// Mitsubishi GX Works2 project: 20151109(変えた)   PLC: Q03UDV

PROGRAM P1
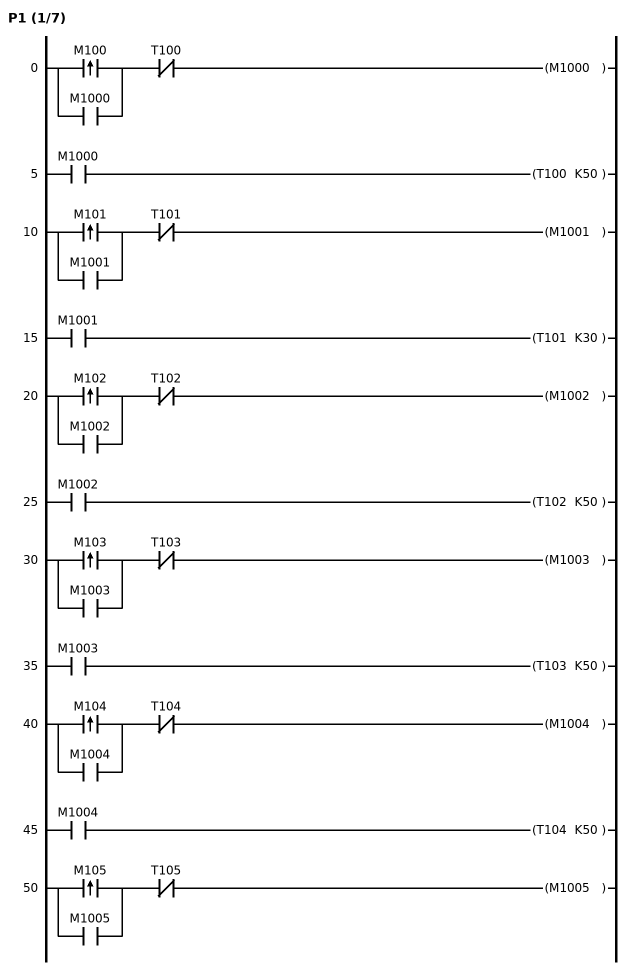
0     LDP     M100
      OR      M1000
      ANI     T100
      OUT     M1000
5     LD      M1000
      OUT     T100 K50
10    LDP     M101
      OR      M1001
      ANI     T101
      OUT     M1001
15    LD      M1001
      OUT     T101 K30
20    LDP     M102
      OR      M1002
      ANI     T102
      OUT     M1002
25    LD      M1002
      OUT     T102 K50
30    LDP     M103
      OR      M1003
      ANI     T103
      OUT     M1003
35    LD      M1003
      OUT     T103 K50
40    LDP     M104
      OR      M1004
      ANI     T104
      OUT     M1004
45    LD      M1004
      OUT     T104 K50
50    LDP     M105
      OR      M1005
      ANI     T105
      OUT     M1005
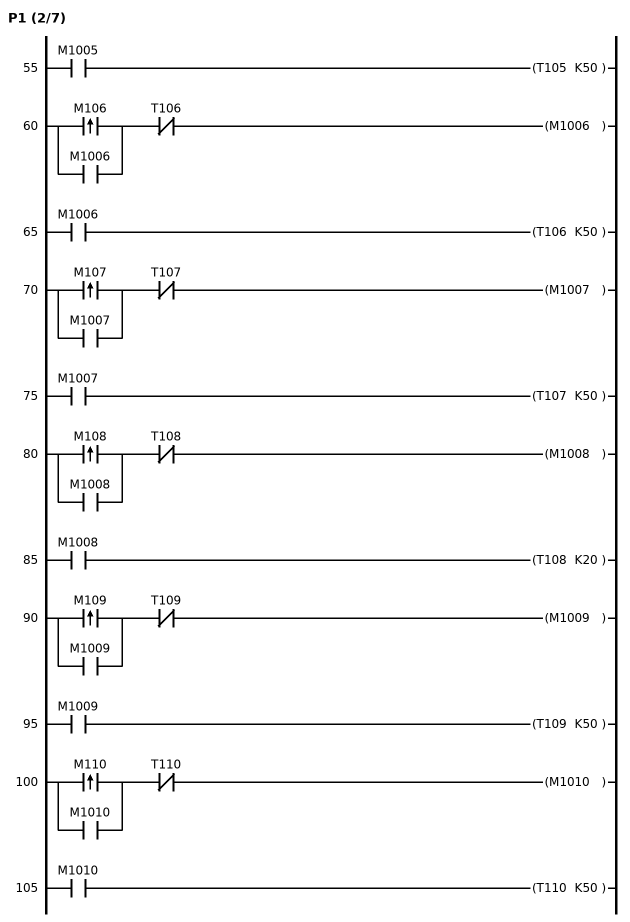
55    LD      M1005
      OUT     T105 K50
60    LDP     M106
      OR      M1006
      ANI     T106
      OUT     M1006
65    LD      M1006
      OUT     T106 K50
70    LDP     M107
      OR      M1007
      ANI     T107
      OUT     M1007
75    LD      M1007
      OUT     T107 K50
80    LDP     M108
      OR      M1008
      ANI     T108
      OUT     M1008
85    LD      M1008
      OUT     T108 K20
90    LDP     M109
      OR      M1009
      ANI     T109
      OUT     M1009
95    LD      M1009
      OUT     T109 K50
100   LDP     M110
      OR      M1010
      ANI     T110
      OUT     M1010
105   LD      M1010
      OUT     T110 K50
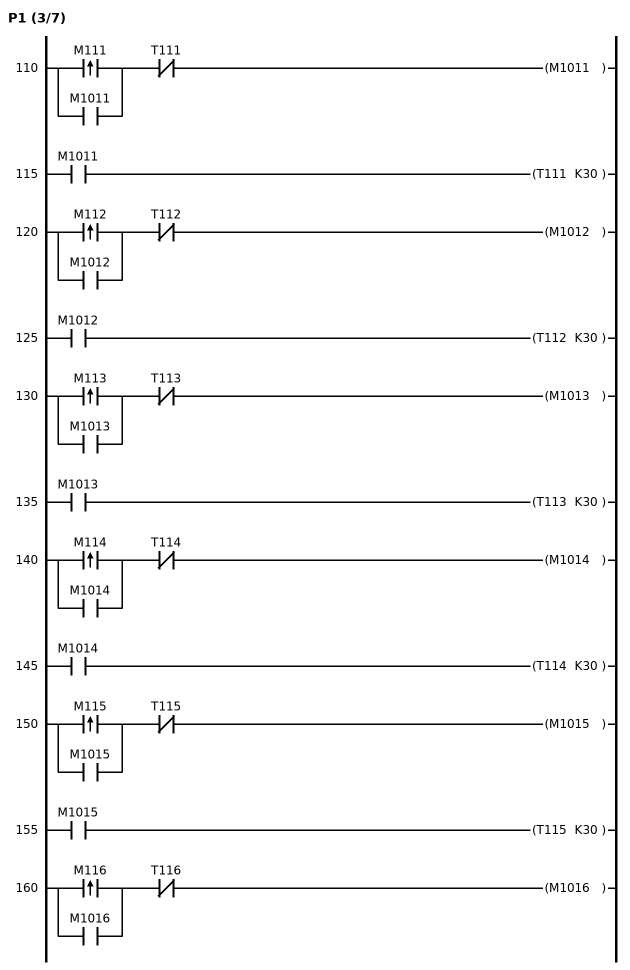
110   LDP     M111
      OR      M1011
      ANI     T111
      OUT     M1011
115   LD      M1011
      OUT     T111 K30
120   LDP     M112
      OR      M1012
      ANI     T112
      OUT     M1012
125   LD      M1012
      OUT     T112 K30
130   LDP     M113
      OR      M1013
      ANI     T113
      OUT     M1013
135   LD      M1013
      OUT     T113 K30
140   LDP     M114
      OR      M1014
      ANI     T114
      OUT     M1014
145   LD      M1014
      OUT     T114 K30
150   LDP     M115
      OR      M1015
      ANI     T115
      OUT     M1015
155   LD      M1015
      OUT     T115 K30
160   LDP     M116
      OR      M1016
      ANI     T116
      OUT     M1016
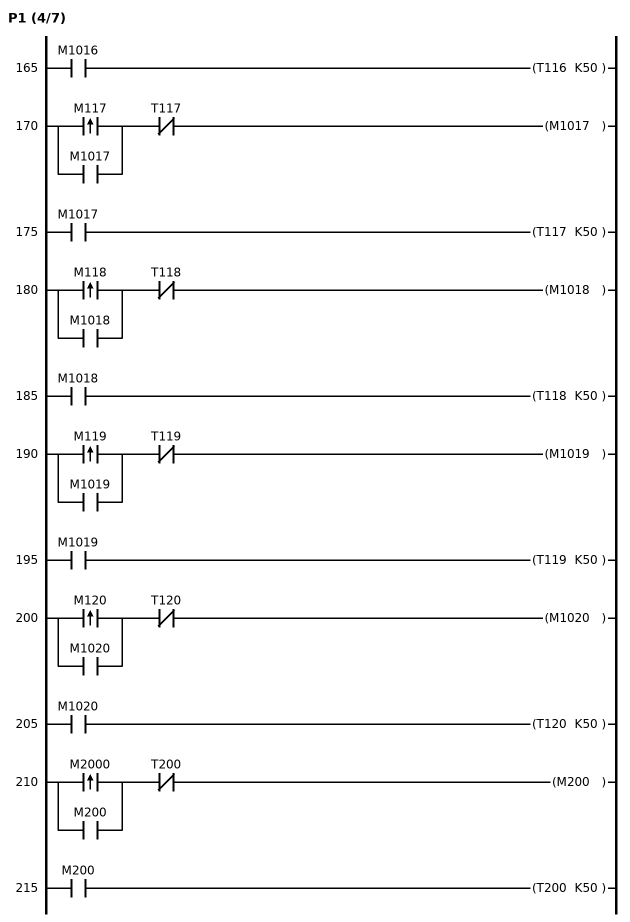
165   LD      M1016
      OUT     T116 K50
170   LDP     M117
      OR      M1017
      ANI     T117
      OUT     M1017
175   LD      M1017
      OUT     T117 K50
180   LDP     M118
      OR      M1018
      ANI     T118
      OUT     M1018
185   LD      M1018
      OUT     T118 K50
190   LDP     M119
      OR      M1019
      ANI     T119
      OUT     M1019
195   LD      M1019
      OUT     T119 K50
200   LDP     M120
      OR      M1020
      ANI     T120
      OUT     M1020
205   LD      M1020
      OUT     T120 K50
210   LDP     M2000
      OR      M200
      ANI     T200
      OUT     M200
215   LD      M200
      OUT     T200 K50
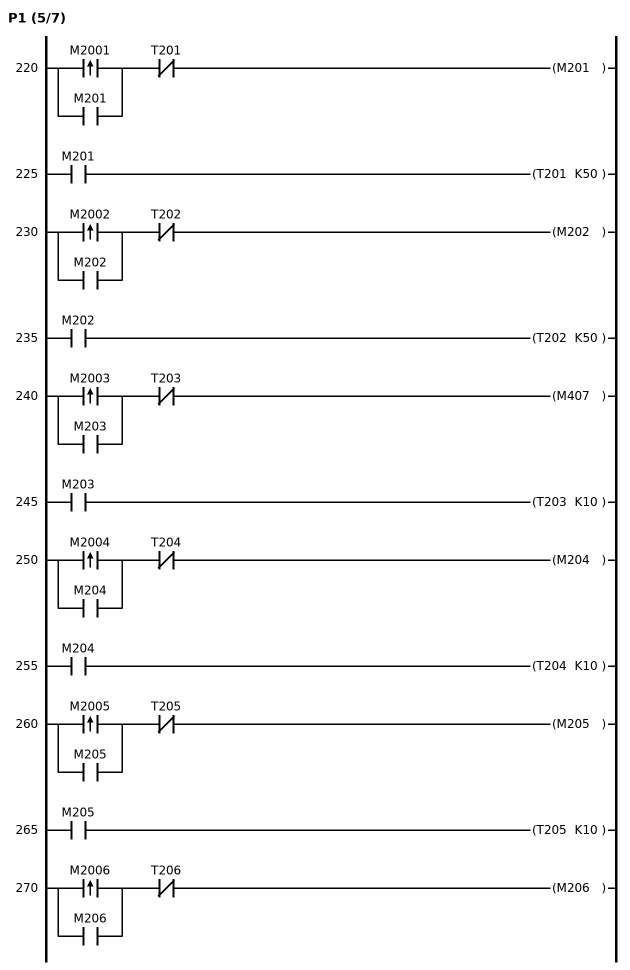
220   LDP     M2001
      OR      M201
      ANI     T201
      OUT     M201
225   LD      M201
      OUT     T201 K50
230   LDP     M2002
      OR      M202
      ANI     T202
      OUT     M202
235   LD      M202
      OUT     T202 K50
240   LDP     M2003
      OR      M203
      ANI     T203
      OUT     M407
245   LD      M203
      OUT     T203 K10
250   LDP     M2004
      OR      M204
      ANI     T204
      OUT     M204
255   LD      M204
      OUT     T204 K10
260   LDP     M2005
      OR      M205
      ANI     T205
      OUT     M205
265   LD      M205
      OUT     T205 K10
270   LDP     M2006
      OR      M206
      ANI     T206
      OUT     M206
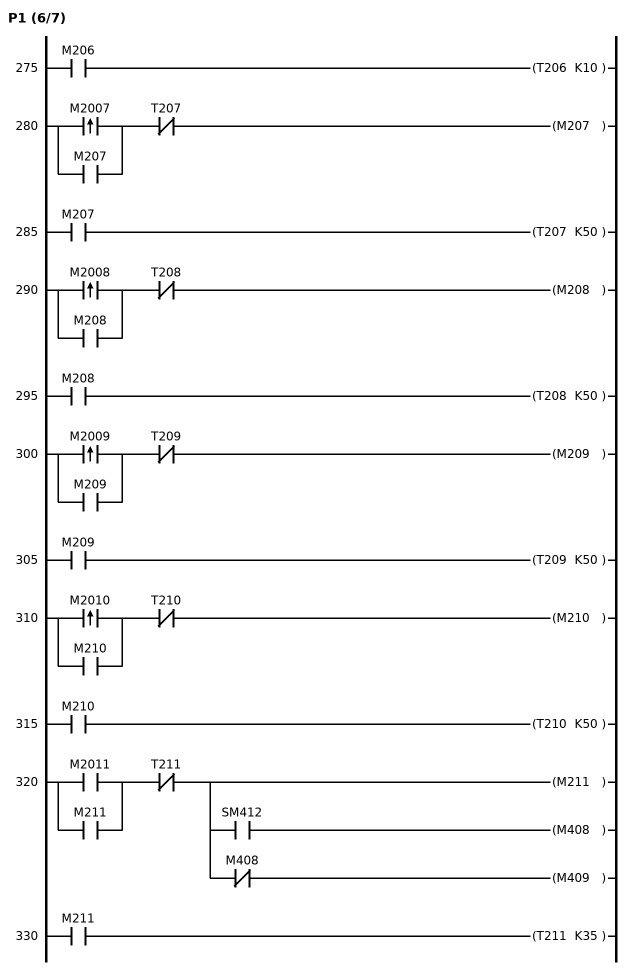
275   LD      M206
      OUT     T206 K10
280   LDP     M2007
      OR      M207
      ANI     T207
      OUT     M207
285   LD      M207
      OUT     T207 K50
290   LDP     M2008
      OR      M208
      ANI     T208
      OUT     M208
295   LD      M208
      OUT     T208 K50
300   LDP     M2009
      OR      M209
      ANI     T209
      OUT     M209
305   LD      M209
      OUT     T209 K50
310   LDP     M2010
      OR      M210
      ANI     T210
      OUT     M210
315   LD      M210
      OUT     T210 K50
320   LD      M2011
      OR      M211
      ANI     T211
      OUT     M211
      MPS
      AND     SM412
      OUT     M408
      MPP
      ANI     M408
      OUT     M409
330   LD      M211
      OUT     T211 K35
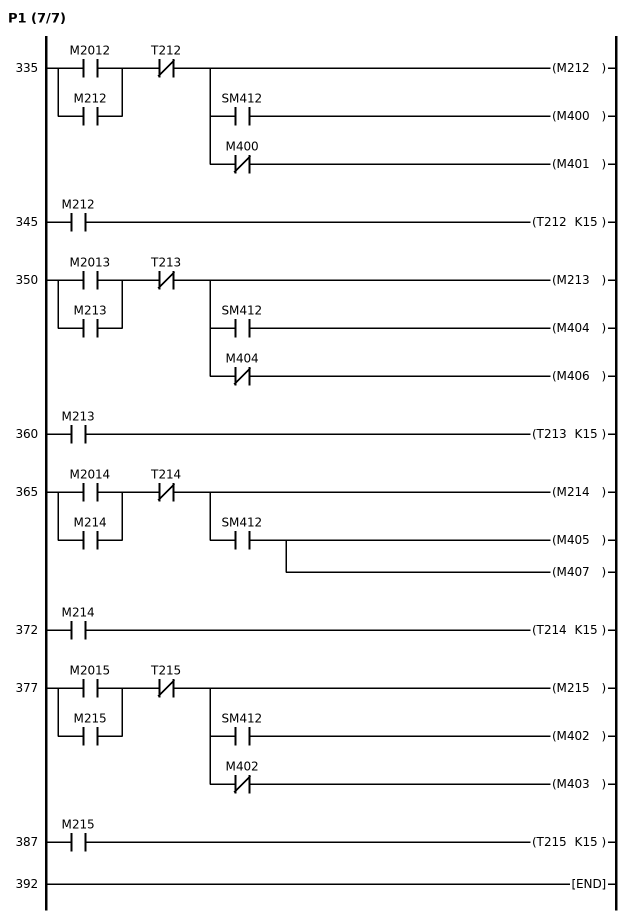
335   LD      M2012
      OR      M212
      ANI     T212
      OUT     M212
      MPS
      AND     SM412
      OUT     M400
      MPP
      ANI     M400
      OUT     M401
345   LD      M212
      OUT     T212 K15
350   LD      M2013
      OR      M213
      ANI     T213
      OUT     M213
      MPS
      AND     SM412
      OUT     M404
      MPP
      ANI     M404
      OUT     M406
360   LD      M213
      OUT     T213 K15
365   LD      M2014
      OR      M214
      ANI     T214
      OUT     M214
      AND     SM412
      OUT     M405
      OUT     M407
372   LD      M214
      OUT     T214 K15
377   LD      M2015
      OR      M215
      ANI     T215
      OUT     M215
      MPS
      AND     SM412
      OUT     M402
      MPP
      ANI     M402
      OUT     M403
387   LD      M215
      OUT     T215 K15
392   END
END_PROGRAM

PROGRAM P2
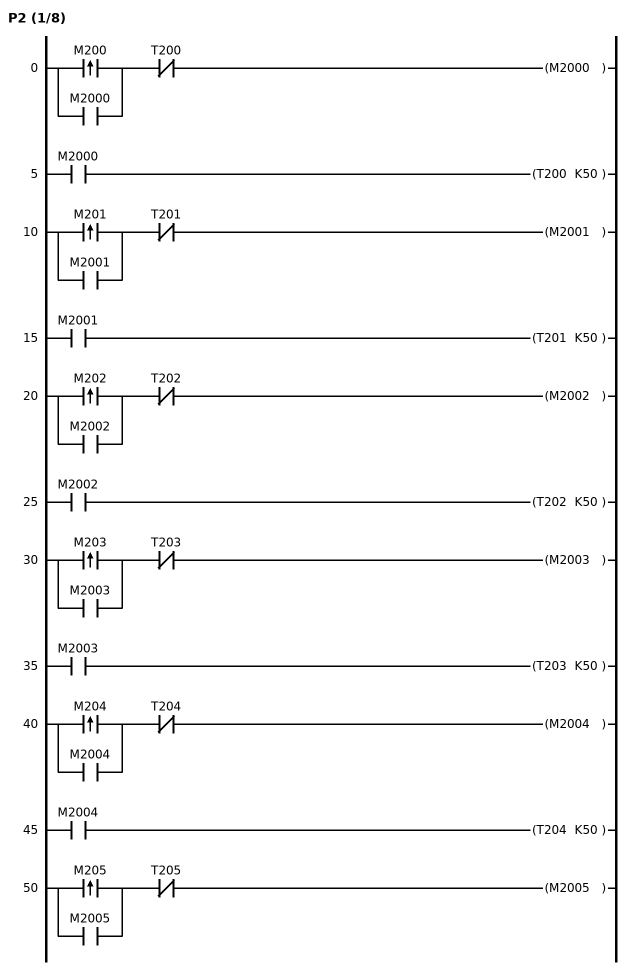
0     LDP     M200
      OR      M2000
      ANI     T200
      OUT     M2000
5     LD      M2000
      OUT     T200 K50
10    LDP     M201
      OR      M2001
      ANI     T201
      OUT     M2001
15    LD      M2001
      OUT     T201 K50
20    LDP     M202
      OR      M2002
      ANI     T202
      OUT     M2002
25    LD      M2002
      OUT     T202 K50
30    LDP     M203
      OR      M2003
      ANI     T203
      OUT     M2003
35    LD      M2003
      OUT     T203 K50
40    LDP     M204
      OR      M2004
      ANI     T204
      OUT     M2004
45    LD      M2004
      OUT     T204 K50
50    LDP     M205
      OR      M2005
      ANI     T205
      OUT     M2005
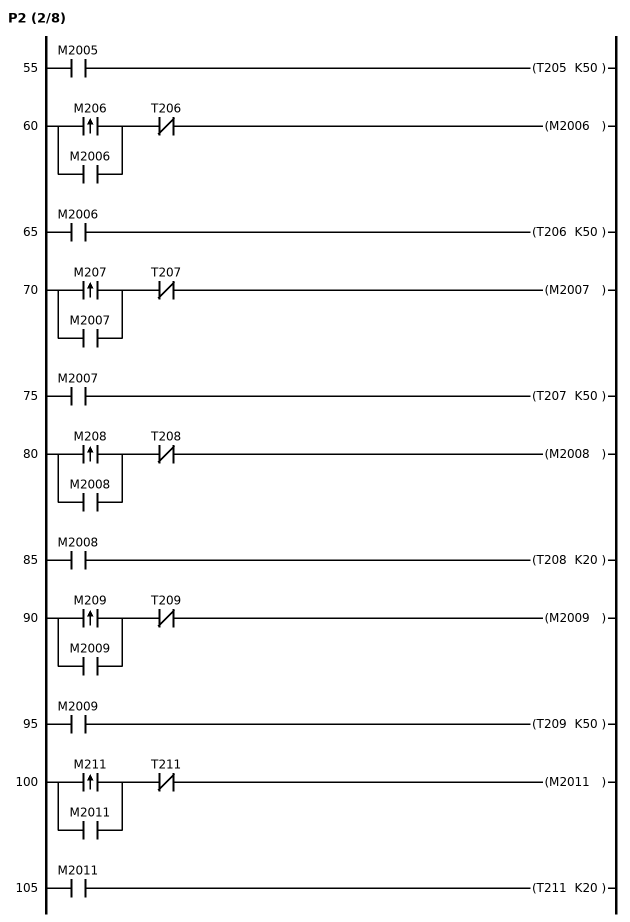
55    LD      M2005
      OUT     T205 K50
60    LDP     M206
      OR      M2006
      ANI     T206
      OUT     M2006
65    LD      M2006
      OUT     T206 K50
70    LDP     M207
      OR      M2007
      ANI     T207
      OUT     M2007
75    LD      M2007
      OUT     T207 K50
80    LDP     M208
      OR      M2008
      ANI     T208
      OUT     M2008
85    LD      M2008
      OUT     T208 K20
90    LDP     M209
      OR      M2009
      ANI     T209
      OUT     M2009
95    LD      M2009
      OUT     T209 K50
100   LDP     M211
      OR      M2011
      ANI     T211
      OUT     M2011
105   LD      M2011
      OUT     T211 K20
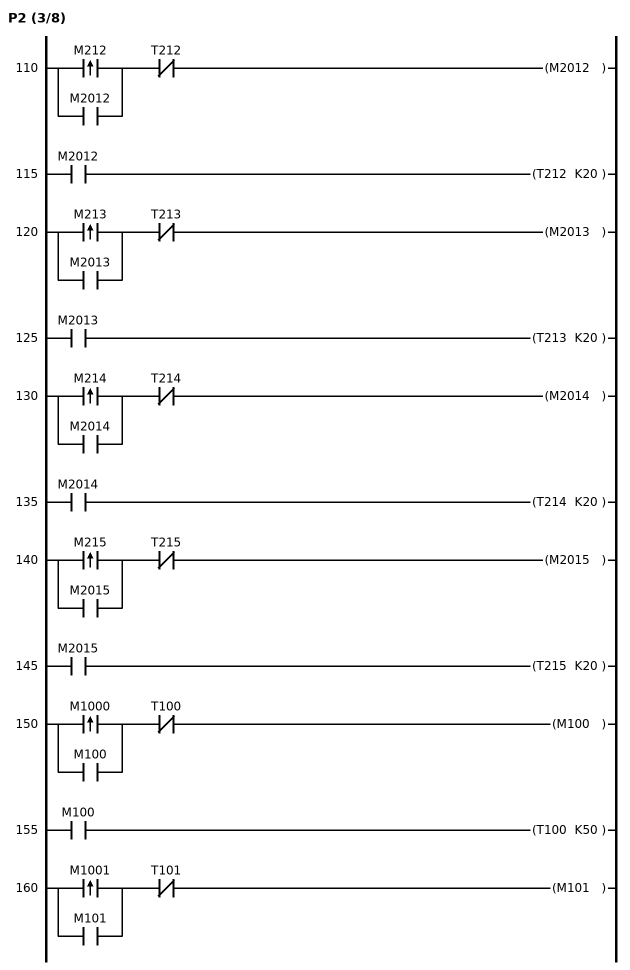
110   LDP     M212
      OR      M2012
      ANI     T212
      OUT     M2012
115   LD      M2012
      OUT     T212 K20
120   LDP     M213
      OR      M2013
      ANI     T213
      OUT     M2013
125   LD      M2013
      OUT     T213 K20
130   LDP     M214
      OR      M2014
      ANI     T214
      OUT     M2014
135   LD      M2014
      OUT     T214 K20
140   LDP     M215
      OR      M2015
      ANI     T215
      OUT     M2015
145   LD      M2015
      OUT     T215 K20
150   LDP     M1000
      OR      M100
      ANI     T100
      OUT     M100
155   LD      M100
      OUT     T100 K50
160   LDP     M1001
      OR      M101
      ANI     T101
      OUT     M101
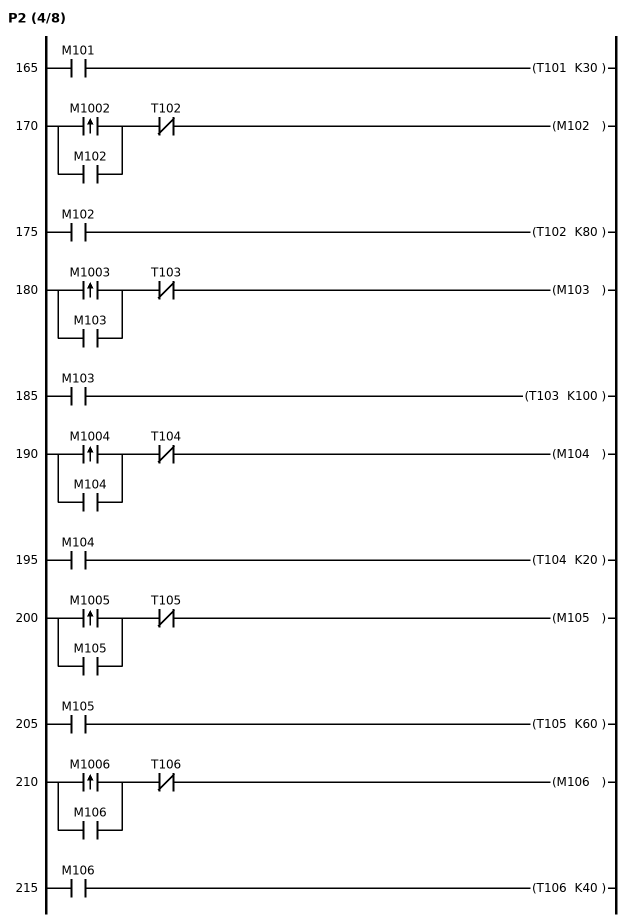
165   LD      M101
      OUT     T101 K30
170   LDP     M1002
      OR      M102
      ANI     T102
      OUT     M102
175   LD      M102
      OUT     T102 K80
180   LDP     M1003
      OR      M103
      ANI     T103
      OUT     M103
185   LD      M103
      OUT     T103 K100
190   LDP     M1004
      OR      M104
      ANI     T104
      OUT     M104
195   LD      M104
      OUT     T104 K20
200   LDP     M1005
      OR      M105
      ANI     T105
      OUT     M105
205   LD      M105
      OUT     T105 K60
210   LDP     M1006
      OR      M106
      ANI     T106
      OUT     M106
215   LD      M106
      OUT     T106 K40
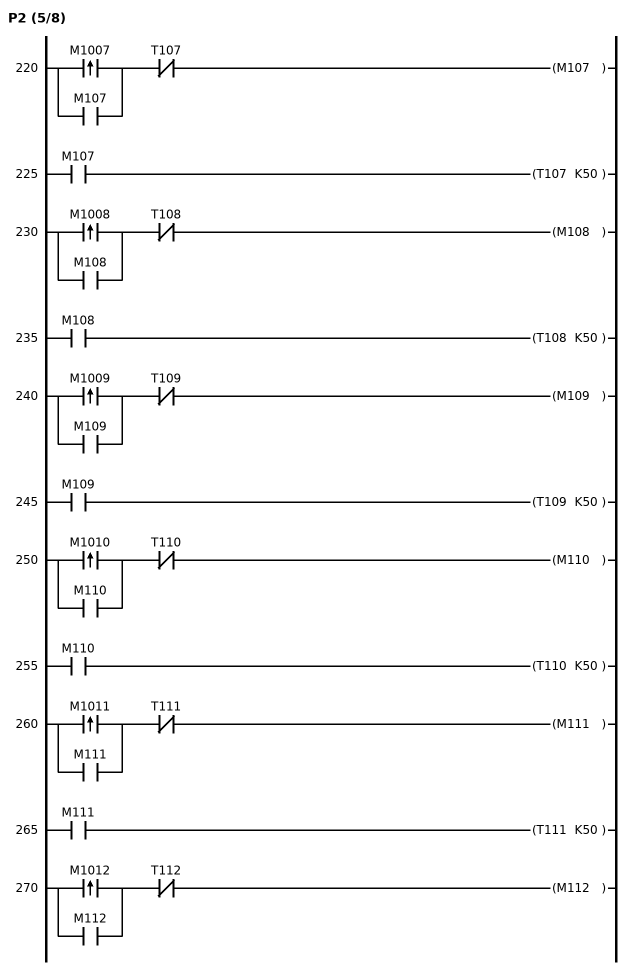
220   LDP     M1007
      OR      M107
      ANI     T107
      OUT     M107
225   LD      M107
      OUT     T107 K50
230   LDP     M1008
      OR      M108
      ANI     T108
      OUT     M108
235   LD      M108
      OUT     T108 K50
240   LDP     M1009
      OR      M109
      ANI     T109
      OUT     M109
245   LD      M109
      OUT     T109 K50
250   LDP     M1010
      OR      M110
      ANI     T110
      OUT     M110
255   LD      M110
      OUT     T110 K50
260   LDP     M1011
      OR      M111
      ANI     T111
      OUT     M111
265   LD      M111
      OUT     T111 K50
270   LDP     M1012
      OR      M112
      ANI     T112
      OUT     M112
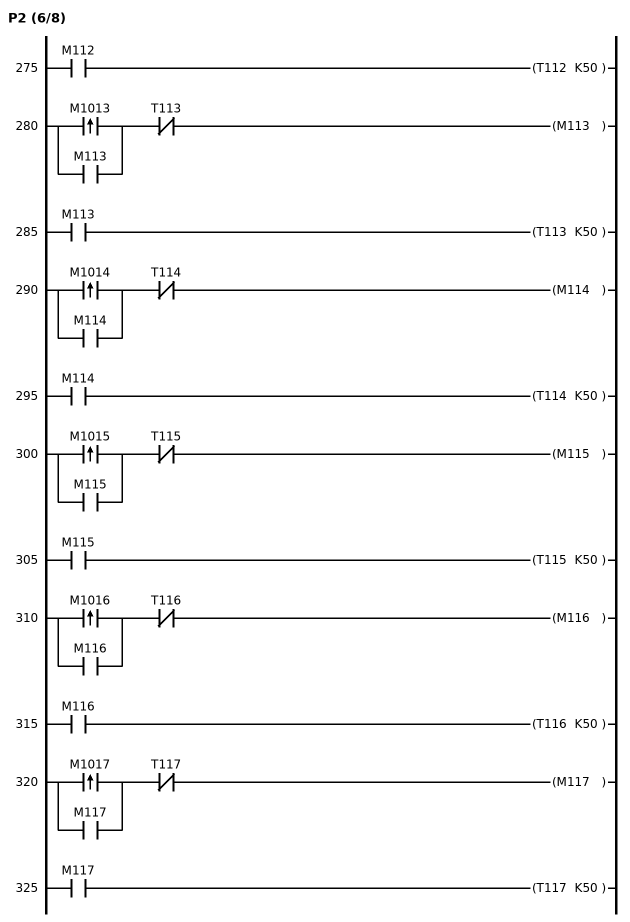
275   LD      M112
      OUT     T112 K50
280   LDP     M1013
      OR      M113
      ANI     T113
      OUT     M113
285   LD      M113
      OUT     T113 K50
290   LDP     M1014
      OR      M114
      ANI     T114
      OUT     M114
295   LD      M114
      OUT     T114 K50
300   LDP     M1015
      OR      M115
      ANI     T115
      OUT     M115
305   LD      M115
      OUT     T115 K50
310   LDP     M1016
      OR      M116
      ANI     T116
      OUT     M116
315   LD      M116
      OUT     T116 K50
320   LDP     M1017
      OR      M117
      ANI     T117
      OUT     M117
325   LD      M117
      OUT     T117 K50
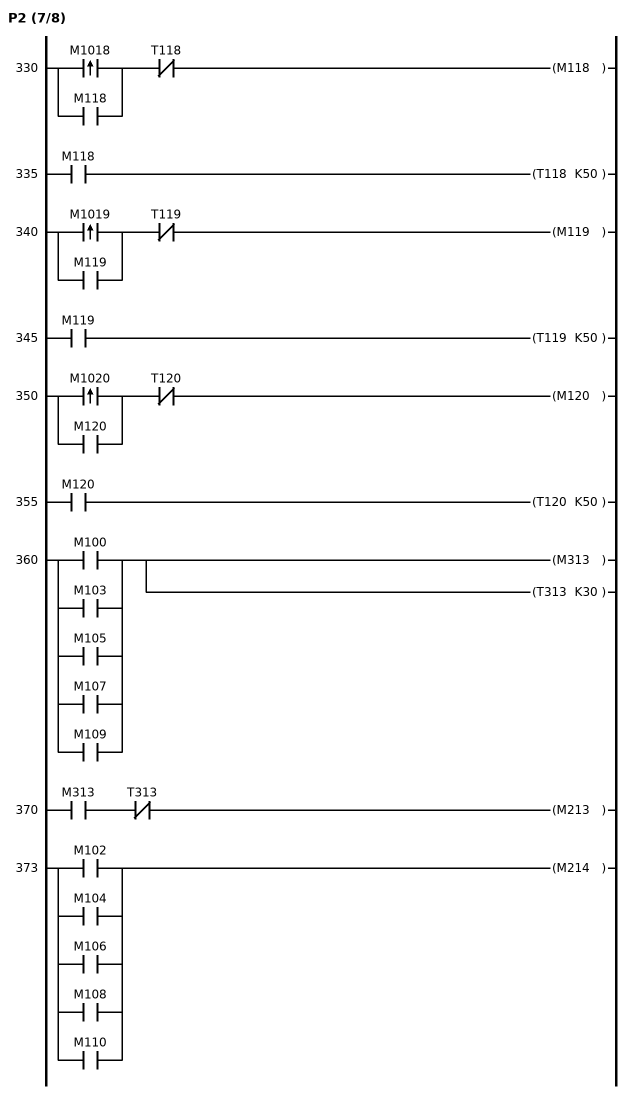
330   LDP     M1018
      OR      M118
      ANI     T118
      OUT     M118
335   LD      M118
      OUT     T118 K50
340   LDP     M1019
      OR      M119
      ANI     T119
      OUT     M119
345   LD      M119
      OUT     T119 K50
350   LDP     M1020
      OR      M120
      ANI     T120
      OUT     M120
355   LD      M120
      OUT     T120 K50
360   LD      M100
      OR      M103
      OR      M105
      OR      M107
      OR      M109
      OUT     M313
      OUT     T313 K30
370   LD      M313
      ANI     T313
      OUT     M213
373   LD      M102
      OR      M104
      OR      M106
      OR      M108
      OR      M110
      OUT     M214
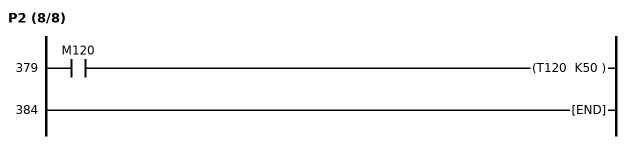
379   LD      M120
      OUT     T120 K50
384   END
END_PROGRAM

PROGRAM P3
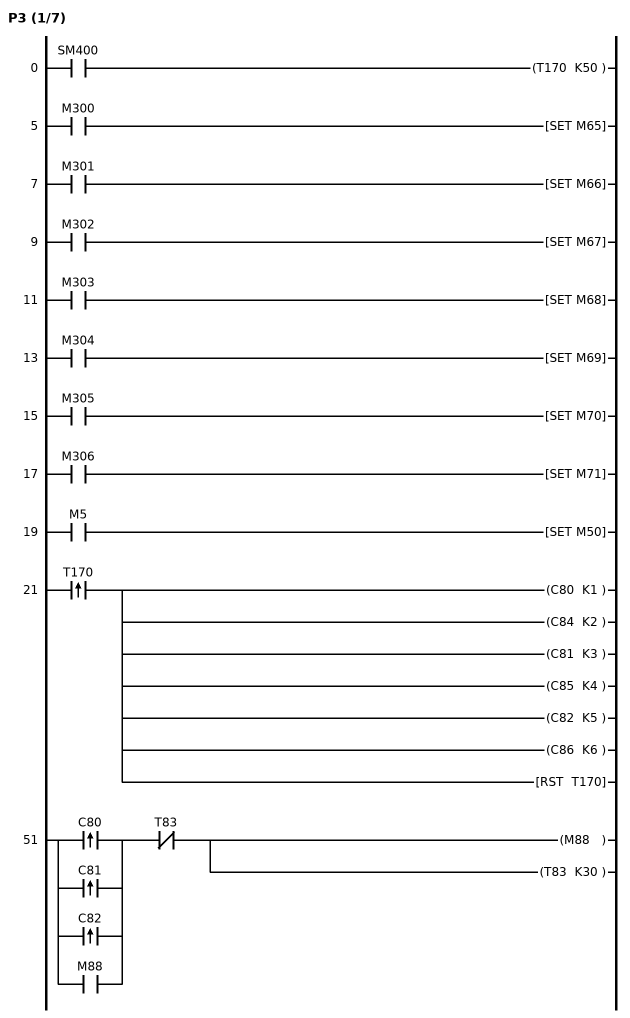
0     LD      SM400
      OUT     T170 K50
5     LD      M300
      SET     M65
7     LD      M301
      SET     M66
9     LD      M302
      SET     M67
11    LD      M303
      SET     M68
13    LD      M304
      SET     M69
15    LD      M305
      SET     M70
17    LD      M306
      SET     M71
19    LD      M5
      SET     M50
21    LDP     T170
      OUT     C80 K1
      OUT     C84 K2
      OUT     C81 K3
      OUT     C85 K4
      OUT     C82 K5
      OUT     C86 K6
      RST     T170
51    LDP     C80
      ORP     C81
      ORP     C82
      OR      M88
      ANI     T83
      OUT     M88
      OUT     T83 K30
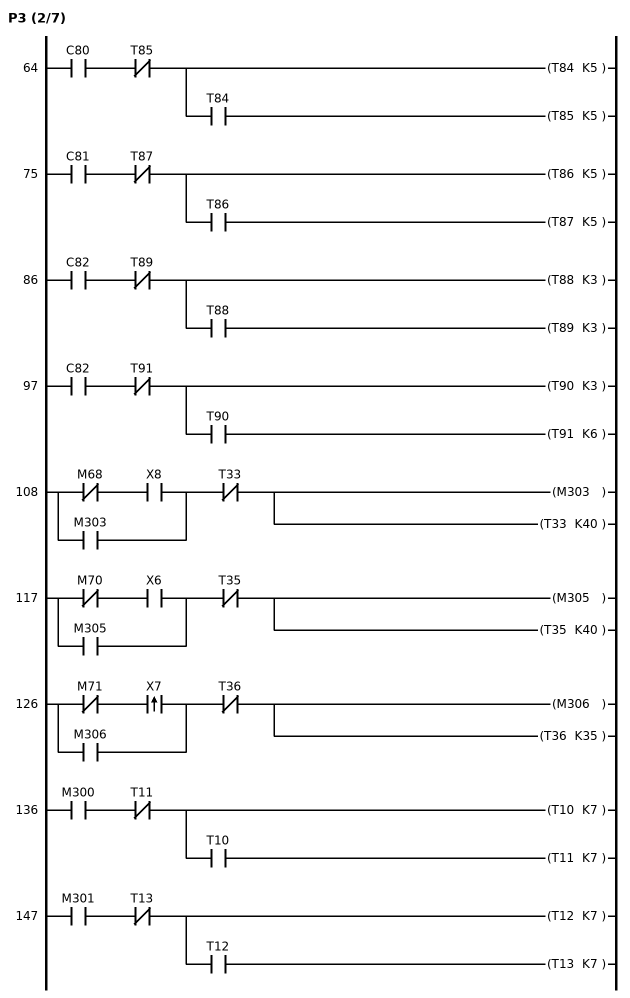
64    LD      C80
      ANI     T85
      OUT     T84 K5
      AND     T84
      OUT     T85 K5
75    LD      C81
      ANI     T87
      OUT     T86 K5
      AND     T86
      OUT     T87 K5
86    LD      C82
      ANI     T89
      OUT     T88 K3
      AND     T88
      OUT     T89 K3
97    LD      C82
      ANI     T91
      OUT     T90 K3
      AND     T90
      OUT     T91 K6
108   LDI     M68
      AND     X8
      OR      M303
      ANI     T33
      OUT     M303
      OUT     T33 K40
117   LDI     M70
      AND     X6
      OR      M305
      ANI     T35
      OUT     M305
      OUT     T35 K40
126   LDI     M71
      ANDP    X7
      OR      M306
      ANI     T36
      OUT     M306
      OUT     T36 K35
136   LD      M300
      ANI     T11
      OUT     T10 K7
      AND     T10
      OUT     T11 K7
147   LD      M301
      ANI     T13
      OUT     T12 K7
      AND     T12
      OUT     T13 K7
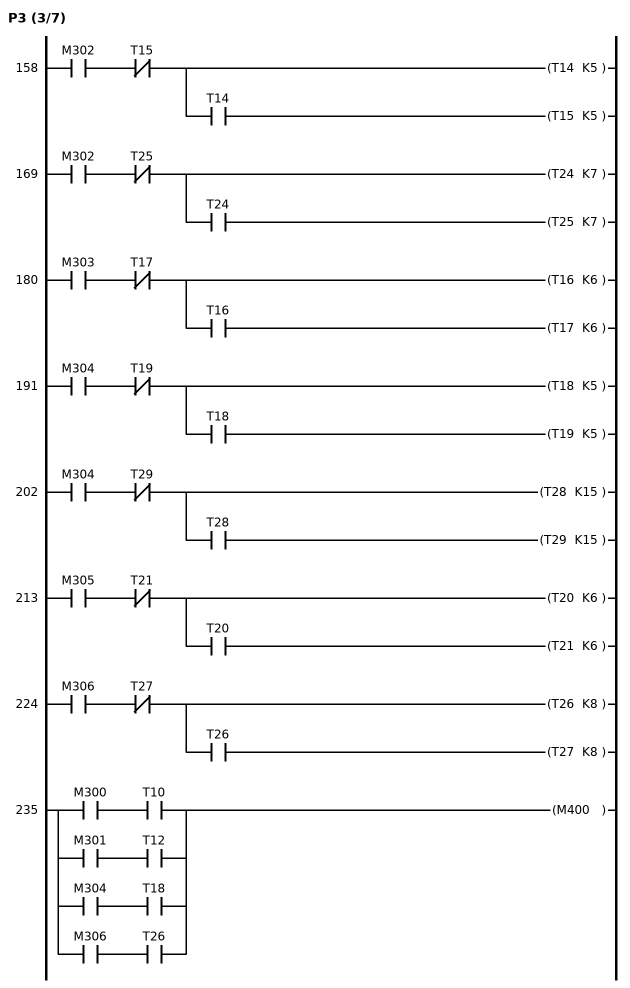
158   LD      M302
      ANI     T15
      OUT     T14 K5
      AND     T14
      OUT     T15 K5
169   LD      M302
      ANI     T25
      OUT     T24 K7
      AND     T24
      OUT     T25 K7
180   LD      M303
      ANI     T17
      OUT     T16 K6
      AND     T16
      OUT     T17 K6
191   LD      M304
      ANI     T19
      OUT     T18 K5
      AND     T18
      OUT     T19 K5
202   LD      M304
      ANI     T29
      OUT     T28 K15
      AND     T28
      OUT     T29 K15
213   LD      M305
      ANI     T21
      OUT     T20 K6
      AND     T20
      OUT     T21 K6
224   LD      M306
      ANI     T27
      OUT     T26 K8
      AND     T26
      OUT     T27 K8
235   LD      M300
      AND     T10
      LD      M301
      AND     T12
      ORB
      LD      M304
      AND     T18
      ORB
      LD      M306
      AND     T26
      ORB
      OUT     M400
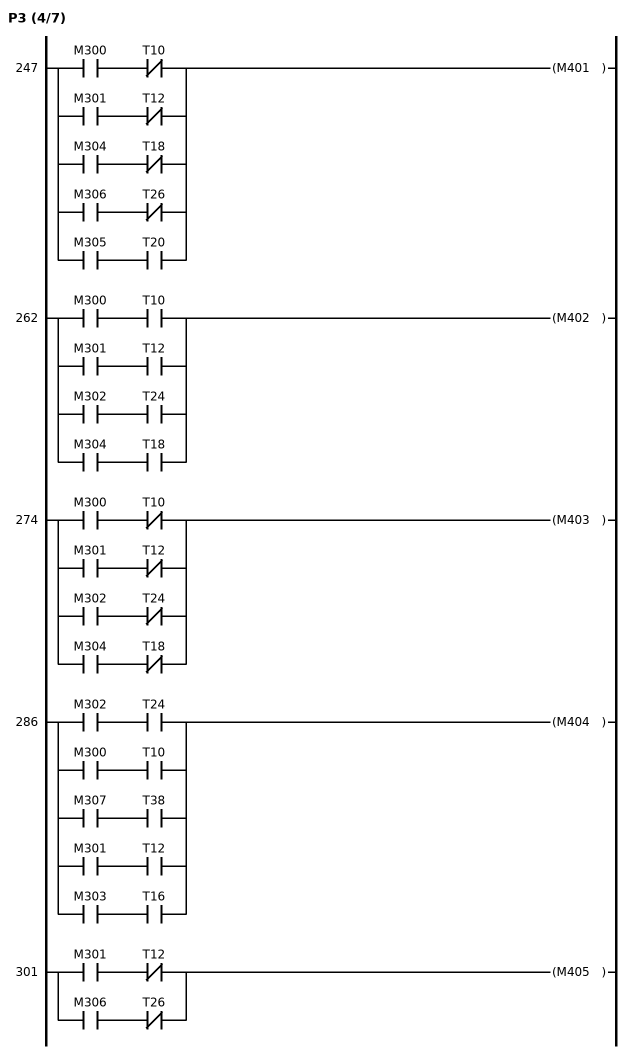
247   LD      M300
      ANI     T10
      LD      M301
      ANI     T12
      ORB
      LD      M304
      ANI     T18
      ORB
      LD      M306
      ANI     T26
      ORB
      LD      M305
      AND     T20
      ORB
      OUT     M401
262   LD      M300
      AND     T10
      LD      M301
      AND     T12
      ORB
      LD      M302
      AND     T24
      ORB
      LD      M304
      AND     T18
      ORB
      OUT     M402
274   LD      M300
      ANI     T10
      LD      M301
      ANI     T12
      ORB
      LD      M302
      ANI     T24
      ORB
      LD      M304
      ANI     T18
      ORB
      OUT     M403
286   LD      M302
      AND     T24
      LD      M300
      AND     T10
      ORB
      LD      M307
      AND     T38
      ORB
      LD      M301
      AND     T12
      ORB
      LD      M303
      AND     T16
      ORB
      OUT     M404
301   LD      M301
      ANI     T12
      LD      M306
      ANI     T26
      ORB
      OUT     M405
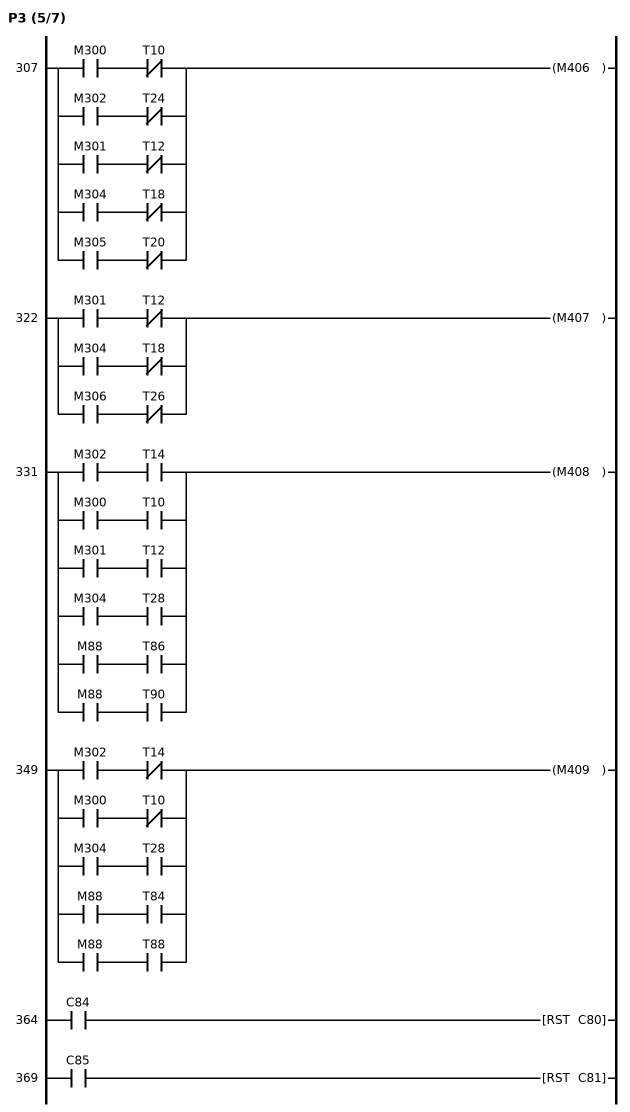
307   LD      M300
      ANI     T10
      LD      M302
      ANI     T24
      ORB
      LD      M301
      ANI     T12
      ORB
      LD      M304
      ANI     T18
      ORB
      LD      M305
      ANI     T20
      ORB
      OUT     M406
322   LD      M301
      ANI     T12
      LD      M304
      ANI     T18
      ORB
      LD      M306
      ANI     T26
      ORB
      OUT     M407
331   LD      M302
      AND     T14
      LD      M300
      AND     T10
      ORB
      LD      M301
      AND     T12
      ORB
      LD      M304
      AND     T28
      ORB
      LD      M88
      AND     T86
      ORB
      LD      M88
      AND     T90
      ORB
      OUT     M408
349   LD      M302
      ANI     T14
      LD      M300
      ANI     T10
      ORB
      LD      M304
      AND     T28
      ORB
      LD      M88
      AND     T84
      ORB
      LD      M88
      AND     T88
      ORB
      OUT     M409
364   LD      C84
      RST     C80
369   LD      C85
      RST     C81
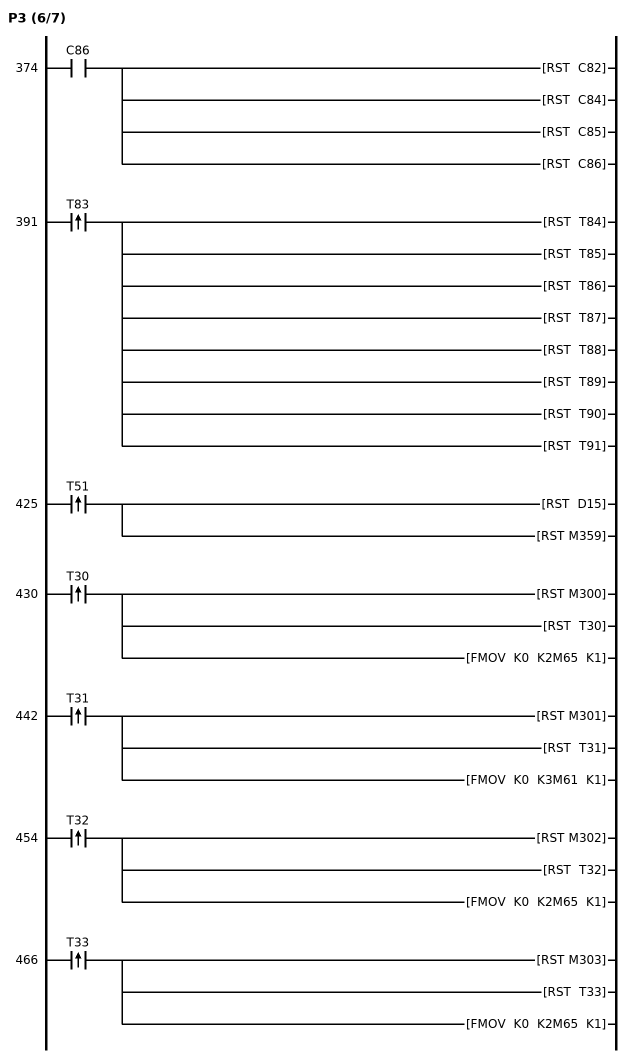
374   LD      C86
      RST     C82
      RST     C84
      RST     C85
      RST     C86
391   LDP     T83
      RST     T84
      RST     T85
      RST     T86
      RST     T87
      RST     T88
      RST     T89
      RST     T90
      RST     T91
425   LDP     T51
      RST     D15
      RST     M359
430   LDP     T30
      RST     M300
      RST     T30
      FMOV    K0 K2M65 K1
442   LDP     T31
      RST     M301
      RST     T31
      FMOV    K0 K3M61 K1
454   LDP     T32
      RST     M302
      RST     T32
      FMOV    K0 K2M65 K1
466   LDP     T33
      RST     M303
      RST     T33
      FMOV    K0 K2M65 K1
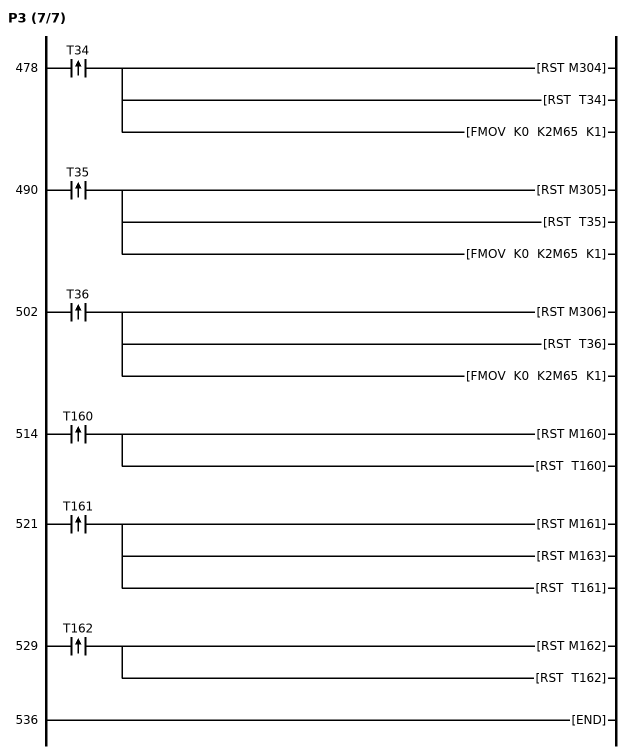
478   LDP     T34
      RST     M304
      RST     T34
      FMOV    K0 K2M65 K1
490   LDP     T35
      RST     M305
      RST     T35
      FMOV    K0 K2M65 K1
502   LDP     T36
      RST     M306
      RST     T36
      FMOV    K0 K2M65 K1
514   LDP     T160
      RST     M160
      RST     T160
521   LDP     T161
      RST     M161
      RST     M163
      RST     T161
529   LDP     T162
      RST     M162
      RST     T162
536   END
END_PROGRAM

PROGRAM P4
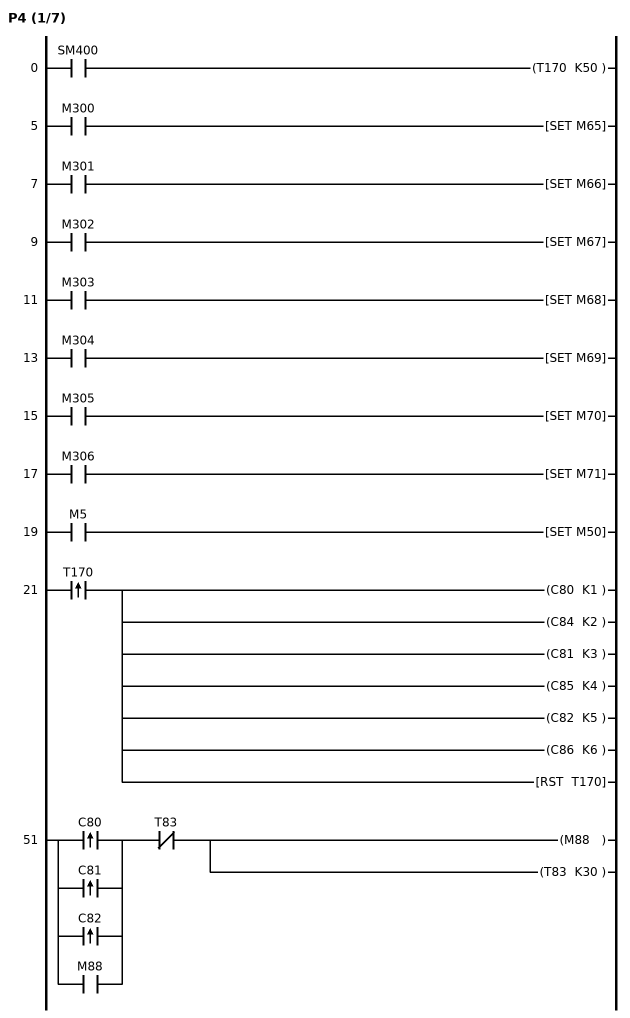
0     LD      SM400
      OUT     T170 K50
5     LD      M300
      SET     M65
7     LD      M301
      SET     M66
9     LD      M302
      SET     M67
11    LD      M303
      SET     M68
13    LD      M304
      SET     M69
15    LD      M305
      SET     M70
17    LD      M306
      SET     M71
19    LD      M5
      SET     M50
21    LDP     T170
      OUT     C80 K1
      OUT     C84 K2
      OUT     C81 K3
      OUT     C85 K4
      OUT     C82 K5
      OUT     C86 K6
      RST     T170
51    LDP     C80
      ORP     C81
      ORP     C82
      OR      M88
      ANI     T83
      OUT     M88
      OUT     T83 K30
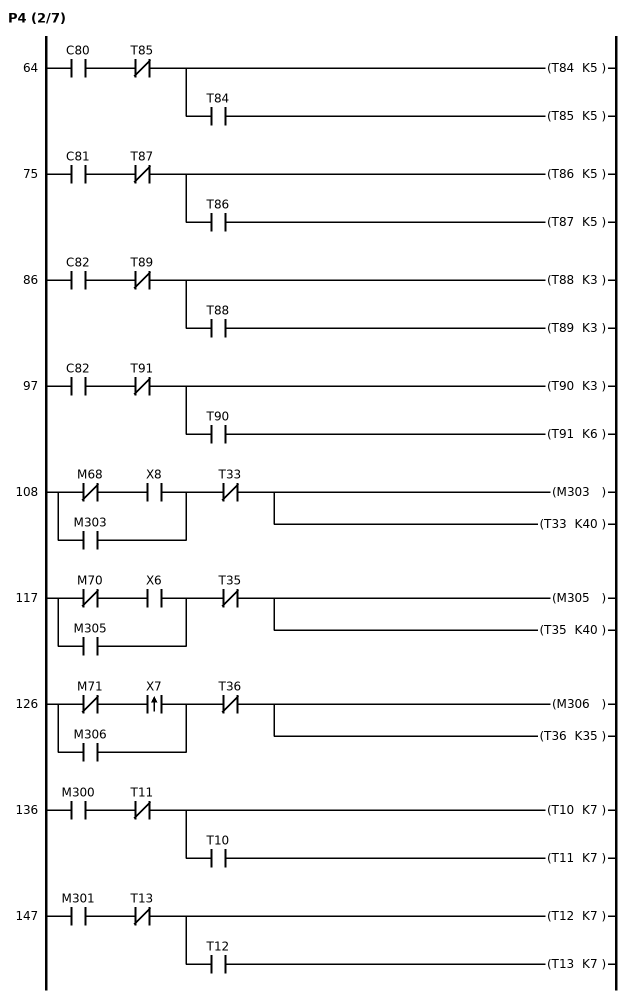
64    LD      C80
      ANI     T85
      OUT     T84 K5
      AND     T84
      OUT     T85 K5
75    LD      C81
      ANI     T87
      OUT     T86 K5
      AND     T86
      OUT     T87 K5
86    LD      C82
      ANI     T89
      OUT     T88 K3
      AND     T88
      OUT     T89 K3
97    LD      C82
      ANI     T91
      OUT     T90 K3
      AND     T90
      OUT     T91 K6
108   LDI     M68
      AND     X8
      OR      M303
      ANI     T33
      OUT     M303
      OUT     T33 K40
117   LDI     M70
      AND     X6
      OR      M305
      ANI     T35
      OUT     M305
      OUT     T35 K40
126   LDI     M71
      ANDP    X7
      OR      M306
      ANI     T36
      OUT     M306
      OUT     T36 K35
136   LD      M300
      ANI     T11
      OUT     T10 K7
      AND     T10
      OUT     T11 K7
147   LD      M301
      ANI     T13
      OUT     T12 K7
      AND     T12
      OUT     T13 K7
